FUNCTION_BLOCK MotorContactor
VAR
	_output	AT%Q*	: BOOL;
END_VAR

METHOD SwitchOff : BOOL
VAR_INPUT
END_VAR
_output := False;
END_METHOD

METHOD SwitchOn : BOOL
VAR_INPUT
END_VAR
_output := True;
END_METHOD

END_FUNCTION_BLOCK

(* stored: Version 1.1.0.1, ProductVersion 3.1.4024.12
   POU MotorContactor: Id {e1462739-47c9-4575-add9-5f065839d072}, SpecialFunc None
   Method SwitchOff: Id {2b0a9879-206a-40e5-8032-7f79867a5df1}
   Method SwitchOn: Id {f96a8c5e-6833-4535-b423-6211447e25fc} *)
